// TwinCAT 3 PLC project Data_Streaming
// ProgramVersion: 3.1.4024.12
// libraries:
//   OSCAT, * (RWTH Aachen University - E.ON Energy Research Center)
//   Tc2_Standard, * (Beckhoff Automation GmbH)
//   Tc2_System, * (Beckhoff Automation GmbH)
//   Tc2_Utilities, * (Beckhoff Automation GmbH)
//   Tc3_IotBase, * (Beckhoff Automation GmbH)
//   Tc3_Module, * (Beckhoff Automation GmbH)
// project tree:
//   DUTs/ ST_Data_Struct.TcDUT
//   GVLs/ Example_CHP.TcGVL, MQTT_Credentials.TcGVL
//   / PlcTask.TcTTO
//   POUs/Components/ BaseComponent.TcPOU, FB_ExampleCHP.TcPOU
//   POUs/Interfaces/ I_Clock.TcIO, I_ImpulseSensor.TcIO, I_TemperatureSensor.TcIO, I_VolumeFlowSensor.TcIO
//   POUs/ MAIN.TcPOU
//   POUs/MQTT/ FB_Get_Unix_Timestamp.TcPOU, FB_Mqtt_Publisher.TcPOU, F_Create_Aedifion_Payload.TcPOU
//   POUs/Sensors/ FB_GasCounter.TcPOU, FB_TempSensPtx.TcPOU, FB_VolSensVmax.TcPOU
// real-time tasks:
//   TASK PlcTask: cycle T#10ms, priority 20, ADS port 350
// I/O:
//   DEVICE SPS (EtherCAT), AmsNetId 5.45.228.127.3.1
//     Klemme 1 (EK1200) [EK1200-5000 EtherCAT Netzteil (2A E-Bus)]
//       Klemme 4 (EL3214) [EL3214 4K. Ana. Eingang PT100 (RTD)]
//       Klemme 3 (EL9011) [EL9011 Endklemme]
// variable links:
//   Data_Streaming/Data_Streaming Instance <-> SPS (EtherCAT)/Term 1 (EK1200)/Term 4 (EL3214)
//     PlcTask Inputs/MAIN.fbCHP.fbChpTin.TempRaw <-> RTD Inputs Channel 1/Value

CONFIGURATION Data_Streaming
    RESOURCE PLC ON TwinCAT3
        TASK PlcTask(INTERVAL := T#10ms, PRIORITY := 20);
        PROGRAM MAIN WITH PlcTask : MAIN;
    END_RESOURCE
END_CONFIGURATION

// ---- DUTs/ST_Data_Struct.TcDUT
TYPE ST_Data_Struct :
	// Datastruct for MQTT messages
STRUCT
	name:STRING(255);
	value:REAL(255);
	topic:STRING(255);
	payload:STRING(255);
	
END_STRUCT
END_TYPE

// ---- GVLs/Example_CHP.TcGVL
{attribute 'qualified_only'}
VAR_GLOBAL
	// CHP - Combined Heat and Power
	
	// Setup MQTT message structs for every reelevant monitoring variable
	
	T_IN:ST_Data_Struct;
	T_IN_name:STRING:='T_sens';	
	T_IN_topic:STRING:='9kfHHUyq';
	
	T_OUT:ST_Data_Struct;
	T_OUT_name:STRING:='bacnet501-NAE01ERC-EBC-4120MONI-AEMW045-TBE-CHP-T-out';	
	T_OUT_topic:STRING:='8Oiu3m3T';
	
	V_dot:ST_Data_Struct;
	V_dot_name:STRING:='bacnet501-NAE01ERC-EBC-4120MONI-AEMW079-TBE-CHP-V-dot';	
	V_dot_topic:STRING:='MNgBovsb';

	V_dot_Gas:ST_Data_Struct;
	V_dot_Gas_name:STRING:='bacnet501-NAE01ERC-EBC-4120MONI-AEMW088-TBE-CHP-V-dot-Gas';	
	V_dot_Gas_topic:STRING:='CoypqcGt';
	
	I_Gas:ST_Data_Struct;
	I_Gas_name:STRING:='bacnet501-NAE01ERC-EBC-4120MONI-AEMW088-TBE-CHP-Imp-Gas';	
	I_Gas_topic:STRING:='KGFsRU7v';
END_VAR

// ---- GVLs/MQTT_Credentials.TcGVL
{attribute 'qualified_only'}
VAR_GLOBAL
	sHostName :STRING := 'mqtt.bawebcontest.aedifion.io'; // Host name 			IP: 116.203.44.193
	nHostPort :UINT:= 8883; // Host port
	sClientId :STRING:= 'CHiLSPS'; // Client ID
	sTopicPrefix :STRING:= 'mtw/BAWebContest_RWTH-Sim/'; // Prefix for every MQTT topic
	nKeepAlive :UINT := 60;      // keep alive time in seconds
	sUserName :STRING:= 'mqtt_bawebcontest_rwth-sim'; // User name
	sUserPassword:STRING := 't5xSVcgWEbc7E4pxKePpumeL07npMt'; // User password
	sTlsVersion:STRING := 'tlsv1.2' ; // TLS version
	sCaPath:STRING:='path/to/file.pem';	// Path to client certificate (on the PLC)
	bNoServerCertCheck:BOOL:=TRUE; // True to check server certificate
END_VAR

// ---- POUs/Interfaces/I_Clock.TcIO
INTERFACE I_Clock
// Interface for every time dependent method

PROPERTY milliseconds : ULINT
GET
END_GET
SET
END_SET
END_PROPERTY

PROPERTY nanoseconds : ULINT
GET
END_GET
SET
END_SET
END_PROPERTY

METHOD Run : BOOL
VAR_INPUT
END_VAR
END_METHOD

PROPERTY seconds : ULINT
GET
END_GET
SET
END_SET
END_PROPERTY

END_INTERFACE

// ---- POUs/Interfaces/I_ImpulseSensor.TcIO
INTERFACE I_ImpulseSensor

PROPERTY nImpulses : UINT
GET
END_GET
SET
END_SET
END_PROPERTY

METHOD Run : BOOL
VAR_INPUT
END_VAR
END_METHOD

END_INTERFACE

// ---- POUs/Interfaces/I_TemperatureSensor.TcIO
INTERFACE I_TemperatureSensor

METHOD Run
VAR_INPUT
END_VAR
END_METHOD

PROPERTY Temperature : REAL
GET
END_GET
SET
END_SET
END_PROPERTY

END_INTERFACE

// ---- POUs/Interfaces/I_VolumeFlowSensor.TcIO
INTERFACE I_VolumeFlowSensor

METHOD Run : BOOL
VAR_INPUT
END_VAR
END_METHOD

PROPERTY VolumeFlow : REAL
GET
END_GET
SET
END_SET
END_PROPERTY

END_INTERFACE

// ---- POUs/MAIN.TcPOU
PROGRAM MAIN
VAR
	//MQTT
	fbMQTT:FB_Mqtt_Publisher; // MQTT publisher
	Connected:BOOL:=FALSE; // Connection status
	// Timing
	i:UDINT; // Counter for every cycle (just to see progress)
	fbTimer:TON:=(PT:=T#20S); // Initialize timer with delay of 20 seconds
	
	// Example Component
	fbCHP:FB_ExampleCHP; // CHP
	
END_VAR

// Connect to MQTT Broker if not already connected
IF Connected=FALSE THEN
	fbMQTT.Connect();
	// Update connection status
	Connected:=fbMQTT.Connected;
END_IF


IF Connected THEN
	fbTimer(IN:=TRUE); // Start timer
	IF fbTimer.Q THEN // If timer reaches delay (20s) start publishing process
		fbTimer(IN:=FALSE); // Reset timer for next cycle
		i := i + 1; // Count cycle
		
		// Publish for every component
		fbCHP.run();
		fbMQTT.Publish_Payload(Example_CHP.T_IN);
		fbMQTT.Publish_Payload(Example_CHP.T_OUT);
		fbMQTT.Publish_Payload(Example_CHP.V_dot);
		fbMQTT.Publish_Payload(Example_CHP.I_Gas);
		fbMQTT.Publish_Payload(Example_CHP.V_dot_Gas);
		
	END_IF
END_IF

END_PROGRAM

// ---- POUs/MQTT/FB_Mqtt_Publisher.TcPOU
FUNCTION_BLOCK FB_Mqtt_Publisher
VAR_INPUT
	
END_VAR
VAR_OUTPUT
END_VAR
VAR
	// Twincat MQTT Client
	fbMqttClient : FB_IotMqttClient; // Enables communication with an MQTT broker
	bSetParameter : BOOL :=	TRUE; // If True, the borker credentials are set in the MQTT client
	bConnect : BOOL	:= TRUE; // If true, the client communicates cyclically with the broker
	bConnected : BOOL := FALSE; // True if connected to Broker
	fbMessageQueue : FB_IotMqttMessageQueue; // Queue for MQTT message, following First-in-First-out
	fbMessage : FB_IotMqttMessage; // MQTT message
	
	hrErrorCode: HRESULT; // Error message, needed for debug purposes
	
	eQoS: TCIOTMQTTQOS := TcIotMqttQos.AtMostOnceDelivery; // Type of QoS
	bRetain: BOOL := FALSE; // True, if broker shall retain messages and send them to new subscribers
	bQueue: BOOL := FALSE; // True, if queue shall be used
	
END_VAR

METHOD Connect : BOOL
VAR_INPUT
END_VAR
// Set Connection Parameters
IF bSetParameter THEN
	bSetParameter  := FALSE;
	fbMqttClient.sHostName := MQTT_Credentials.sHostName;
	fbMqttClient.nHostPort := MQTT_Credentials.nHostPort;
	fbMqttClient.sClientId := MQTT_Credentials.sClientId; 
	fbMqttClient.sTopicPrefix := MQTT_Credentials.sTopicPrefix; 
	fbMqttClient.nKeepAlive := MQTT_Credentials.nKeepAlive; 
	fbMqttClient.sUserName := MQTT_Credentials.sUserName ;
	fbMqttClient.sUserPassword := MQTT_Credentials.sUserPassword; 
	// fbMqttClient.stTLS.sVersion := MQTT_Credentials.sTlsVersion;
	// fbMqttClient.stTLS.sCA := MQTT_Credentials.sCaPath;
	// fbMqttClient.stTLS.bNoServerCertCheck := MQTT_Credentials.bNoServerCertCheck;
END_IF

// Connect to broker
fbMqttClient.Execute(bConnect);

// Set connected to true
bConnected:=fbMqttClient.bConnected;
END_METHOD

PROPERTY Connected : BOOL
GET
Connected:=THIS^.bConnected;
END_GET
SET
THIS^.bConnected:=Connected;
END_SET
END_PROPERTY

METHOD Publish_Payload : BOOL
VAR_INPUT
	Datapoint : ST_Data_Struct; // Datapoint in MQTT data truct format
END_VAR
// Publish payload
fbMqttClient.Publish( sTopic:= Datapoint.topic,
pPayload:= ADR(Datapoint.payload), nPayloadSize:= LEN2(ADR(Datapoint.payload))+1,
eQoS:= eQoS, bRetain:= bRetain,
bQueue:= bQueue );
END_METHOD

END_FUNCTION_BLOCK

// ---- POUs/Components/FB_ExampleCHP.TcPOU
FUNCTION_BLOCK FB_ExampleCHP EXTENDS BaseComponent
// This implements a SPECIFIC CHP, this means the following values have to be adjusted, according to each CHP
VAR_INPUT
END_VAR
VAR_OUTPUT
END_VAR
VAR
	// Temperature sensors
	fbChpTin: FB_TempSensPTx(Ptx:=1000);
	fbChpTout: FB_TempSensPTx(Ptx:=1000);
	
	// Volume Flow Sensors
	fbChpVdot: FB_VolSensVmax(Qminimum:=0, Qmaximum:=50, nIntMaximum:=32767, nIntMinimum:=0);
	
	// Gas Counter
	fbGasCHP: FB_GasCounter(fChpGasVtotal:=67868.4, fChpGasImpulse:=0.1);
	
	// Time
	fbUnixTime: FB_Get_Unix_Timestamp;
	ntimestamp: ULINT;
END_VAR

METHOD Run : BOOL
VAR_INPUT
END_VAR
// Start every sensor that is connected
fbChpTin.Run();
fbChpTout.Run();
fbChpVdot.Run();
fbGasCHP.Run();

//TempSensors
Example_CHP.T_IN.value:=fbChpTin.Temperature;
Example_CHP.T_IN.name:=Example_CHP.T_IN_name;
Example_CHP.T_IN.topic:=Example_CHP.T_IN_topic;

Example_CHP.T_OUT.value:=fbChpTout.Temperature;
Example_CHP.T_OUT.name:=Example_CHP.T_OUT_name;
Example_CHP.T_OUT.topic:=Example_CHP.T_OUT_topic;

//Volume Flow Sensor
Example_CHP.V_dot.value:=fbChpVdot.VolumeFlow;
Example_CHP.V_dot.name:=Example_CHP.V_dot_name;
Example_CHP.V_dot.topic:=Example_CHP.V_dot_topic;

//Gas Counter
Example_CHP.I_Gas.value:=fbGasCHP.nImpulses; // Count number of Impulses
Example_CHP.I_Gas.name:=Example_CHP.I_Gas_name;
Example_CHP.I_Gas.topic:=Example_CHP.I_Gas_topic;

Example_CHP.V_dot_Gas.value:=fbGasCHP.fValue; // Add amount of gas per impulse to the initial value
Example_CHP.V_dot_Gas.name:=Example_CHP.V_dot_Gas_name;
Example_CHP.V_dot_Gas.topic:=Example_CHP.V_dot_Gas_topic;

//Get timestamp
fbUnixTime.Run();
ntimestamp:=fbUnixTime.nanoseconds;

//Write Payload
Example_CHP.T_IN.payload:=F_Create_Aedifion_Payload(Example_CHP.T_IN,ntimestamp);
Example_CHP.T_OUT.payload:=F_Create_Aedifion_Payload(Example_CHP.T_OUT,ntimestamp);
Example_CHP.V_dot.payload:=F_Create_Aedifion_Payload(Example_CHP.V_dot,ntimestamp);

Example_CHP.I_Gas.payload:=F_Create_Aedifion_Payload(Example_CHP.I_Gas,ntimestamp);
Example_CHP.V_dot_Gas.payload:=F_Create_Aedifion_Payload(Example_CHP.V_dot_Gas,ntimestamp);
END_METHOD

END_FUNCTION_BLOCK

// ---- POUs/Components/BaseComponent.TcPOU
FUNCTION_BLOCK BaseComponent
VAR_INPUT
END_VAR
VAR_OUTPUT
END_VAR
VAR
	// Time
	ComponentTime: FB_Get_Unix_Timestamp;
	timestamp: ULINT;
END_VAR

METHOD Run : BOOL
VAR_INPUT
END_VAR
END_METHOD

END_FUNCTION_BLOCK

// ---- POUs/MQTT/FB_Get_Unix_Timestamp.TcPOU
FUNCTION_BLOCK FB_Get_Unix_Timestamp IMPLEMENTS I_Clock
// Turns windows systemtime into unix systemtime
VAR_OUTPUT
END_VAR
VAR
	nSeconds: ULINT; // Seconds
    nMilliseconds: ULINT; // Milliseconds
	nNanoseconds: ULINT; // Nanoseconds

	localSystemTime: FB_LocalSystemTime := ( bEnable := TRUE, dwCycle := 1 ); // Time (local time) in system time format
    getTimeZoneInformation: FB_GetTimeZoneInformation; // Gets time zone information
    timeZoneInformation: ST_TimeZoneInformation; // Struct to store information about the timezone
    specificLocalTimeToFileTime: FB_TzSpecificLocalTimeToFileTime; // Converts local time to UTC time
    fileTime: T_FILETIME; // Time (UTC) in file format
    onZerothSecondLastCycle: BOOL; // Variable to track the zeroth second of every cycle
END_VAR

PROPERTY milliseconds : ULINT
GET
milliseconds:=THIS^.nMilliseconds;
END_GET
SET
THIS^.nMilliseconds:=milliseconds;
END_SET
END_PROPERTY

PROPERTY nanoseconds : ULINT
GET
nanoseconds:=THIS^.nNanoseconds;
END_GET
SET
THIS^.nNanoseconds:=nanoseconds;
END_SET
END_PROPERTY

METHOD Run : BOOL
VAR_INPUT
END_VAR
// Get local system time
localSystemTime();

// If first cycle or if its the zeroth second of each minute, the timezone information is updated/synced
IF (timeZoneInformation.standardName = '' OR (localSystemTime.systemTime.wSecond = 0 AND NOT onZerothSecondLastCycle)) THEN
    // Sync timezone information
	getTimeZoneInformation(sNetID := '', bExecute := TRUE, tzInfo => timeZoneInformation);
END_IF;

// Convert local system time to unix timestamps
specificLocalTimeToFileTime(in := SYSTEMTIME_TO_FILETIME(localSystemTime.systemTime), tzInfo := timeZoneInformation, out => fileTime);
// PLC uses Windows systemtime while aedifion needs Linux systemtime. Therefore, the time is converted with 11644473600 seconds
// fileTime contains the timestamp in 2 separate 32-bit objects. With SHL the significant (high) one ist transformed int 64-bit and the less significant 
// one (low) is added to that.
nSeconds := (SHL(DWORD_TO_ULINT(fileTime.dwHighDateTime), 32) + DWORD_TO_ULINT(fileTime.dwLowDateTime)) / 10000000 - 11644473600;
nMilliseconds := nSeconds*1000;
nNanoseconds := nMilliseconds*1000000;

// The zeroth second is reached, the zone information is updated/synced
onZerothSecondLastCycle := localSystemTime.systemTime.wSecond = 0;
END_METHOD

PROPERTY seconds : ULINT
GET
Seconds:=THIS^.nSeconds;
END_GET
SET
THIS^.nSeconds:=Seconds;
END_SET
END_PROPERTY

END_FUNCTION_BLOCK

// ---- POUs/Sensors/FB_TempSensPtx.TcPOU
FUNCTION_BLOCK FB_TempSensPtx IMPLEMENTS I_TemperatureSensor
(*Classic Pt temperature sensor. The ConvFac defines the resulting Pt sensor (i.e. ConvFac=100 -> Pt100).
Measurement is directly converted into °C.*)
VAR_OUTPUT
END_VAR
VAR
	ConvFac : INT := 10; // Conversion factor (for Pt100 this is 100, Pt1000 it`s 1000, ..)
	fTemperature : REAL; // Properties
	TempRaw AT %I* : INT; // Raw value
END_VAR

METHOD FB_init : BOOL
VAR_INPUT
	bInitRetains : BOOL; // if TRUE, the retain variables are initialized (warm start / cold start)
	bInCopyCode : BOOL;  // if TRUE, the instance afterwards gets moved into the copy code (online change)
	Ptx : INT := 100; // x value (for Pt100 this is 100, Pt1000 it`s 1000, ..)
END_VAR
ConvFac := Ptx/10; // Divide by ten to get conversion factor
END_METHOD

METHOD Run
fTemperature := INT_TO_REAL(TempRaw)/ConvFac; // Read and convert raw temperature measurement
END_METHOD

PROPERTY Temperature : REAL
GET
Temperature := THIS^.fTemperature;
END_GET
SET
END_SET
END_PROPERTY

END_FUNCTION_BLOCK

// ---- POUs/Sensors/FB_VolSensVmax.TcPOU
FUNCTION_BLOCK FB_VolSensVmax IMPLEMENTS  I_VolumeFlowSensor
(*Volume flow sensor with minimal and maximal measurement values.
The unit of the returned measurement depends on the unit given in Q_max and Q_min.*)
VAR
	// Conversion Factors for volume flow value
	Q_max: REAL:=5/12; // Maximum acutal value of volume flow sensor measurement
	Q_min: REAL:=0; // Minimum acutal value of volume flow sensor measurement
	// Conversion factors for sensor signal
	nIntMax: INT:=32767; // Maximum digital value of volume flow sensor (this is dependet on the type of volume sensor, check the data sheet)
	nIntMin: INT:=0; // Minimum digital value of volume flow sensor (this is dependet on the type of volume sensor, check the data sheet)

	fVolFlow: REAL; // Property
	nVolFlowRaw AT %I* : INT; // Raw value
END_VAR

METHOD FB_init : BOOL
VAR_INPUT
	bInitRetains : BOOL; // if TRUE, the retain variables are initialized (warm start / cold start)
	bInCopyCode : BOOL;  // if TRUE, the instance afterwards gets moved into the copy code (online change)
	// Conversion Factors for volume flow value
	Qmaximum: REAL:=5/12; // Maximum acutal value of volume flow sensor measurement
	Qminimum: REAL:=0; // Minimum acutal value of volume flow sensor measurement
	// Conversion factors for sensor signal
	nIntMaximum: INT:=32767; // Maximum digital value of volume flow sensor (this is dependet on the type of volume sensor, check the data sheet)
	nIntMinimum: INT:=0; // Minimum digital value of volume flow sensor (this is dependet on the type of volume sensor, check the data sheet)
END_VAR
Q_max:=Qmaximum;
Q_min:=Qminimum;
nIntMax:=nIntMaximum;
nIntMin:=nIntMinimum;
END_METHOD

METHOD Run: BOOL
fVolFlow:=Q_min+INT_TO_REAL(nVolFlowRaw-nIntMin)/(nIntMax-nIntMin)*(Q_max-Q_min); // Convert digital signal to volumeflow values
END_METHOD

PROPERTY VolumeFlow : REAL
GET
VolumeFlow := THIS^.fVolFlow;
END_GET
SET
THIS^.fVolFlow:=VolumeFlow;
END_SET
END_PROPERTY

END_FUNCTION_BLOCK

// ---- POUs/Sensors/FB_GasCounter.TcPOU
FUNCTION_BLOCK FB_GasCounter IMPLEMENTS  I_ImpulseSensor
(*The impulse sensor counts impulses on the input devices. This can be used for gas counter, which trigger cyclic impulses every time a certain 
amount of gas has passed.
Example for a gas counter:
To calculate the total amount of consumed gas of the connected gas counter, firstly the counter at the start of the monitoring process is needed.
Then you can add the amount of gas that triggers the impulse of the gas counter (e.g. 0.1 m³) multiplied with nImpulse to get an approximation of
the current gas counter value*)
VAR
	fChpGasVtot: REAL:=67868.4; // Initial value of gas counter at start of monitoring
	fChpGasImp: REAL:=0.1; // Amount of gas, that triggers the impulse sensor
	nImpulse: UINT := 0; // Current number of registered Impulses
	fValue: REAL := fChpGasVtot; // Current value of gas counter
	nOn AT %I* : BIT; // Input signal of impulse sensor (if set from FALSE to TRUE, nImpulse increases by one)
	Counter: CTU; // Counter object
END_VAR

METHOD FB_init : BOOL
VAR_INPUT
	bInitRetains : BOOL; // if TRUE, the retain variables are initialized (warm start / cold start)
	bInCopyCode : BOOL;  // if TRUE, the instance afterwards gets moved into the copy code (online change)
	fChpGasVtotal: REAL:=67868.4; // Initial value of gas counter at start of monitoring
	fChpGasImpulse: REAL:=0.1; // Amount of gas, that triggers the impulse sensor
END_VAR
fChpGasVtot:=fChpGasVtotal;
fChpGasImp:=fChpGasImpulse;
END_METHOD

PROPERTY nImpulses : UINT
GET
nImpulses := THIS^.nImpulse;
END_GET
SET
 THIS^.nImpulse:=nImpulses;
END_SET
END_PROPERTY

METHOD Run: BOOL
Counter(CU:=nOn); // Count up (if nOn is set from FALSE to TRUE)
nImpulse:=WORD_TO_UINT(Counter.CV); // Write current counter value as UINT
fValue:=fCHPGasVtot+nImpulse*fChpGasImp;
END_METHOD

END_FUNCTION_BLOCK

// ---- POUs/MQTT/F_Create_Aedifion_Payload.TcPOU
FUNCTION F_Create_Aedifion_Payload : STRING(255)
// Creates the payload for aedifion based on the ST_Data_Struct
VAR_INPUT
	Payload:ST_Data_Struct; // MQTT datastruct
	TimeStamp:ULINT; // Timestamp as integer in Nanoseconds
END_VAR
VAR

	timestring:STRING(255); // Temporary variable
	value:STRING(255); // Temporary variable
	msg_1:STRING(255); // Final payload
	msg_2:STRING(255); // Temporary variable
	a:STRING(255):=' '; // String variable for spaces in payload
	b:STRING(255):='value='; // String variable for test in payload
	
END_VAR

// Create strings
timestring:=ULINT_TO_STRING(TimeStamp);
value:=REAL_TO_STRING(Payload.value);

// Concanate message
msg_1:=CONCAT(Payload.name,a);
msg_2:=CONCAT(msg_1,b);
msg_1:=CONCAT(msg_2,value);
msg_2:=CONCAT(msg_1,a);
msg_1:=CONCAT(msg_2,timestring);


F_Create_Aedifion_Payload:=msg_1;

END_FUNCTION
